METHOD _log : BOOL
  VAR_INPUT
    {attribute 'TcHmiSymbol.Show'}
    name : STRING;  (* Name of this function block instance *)
  END_VAR
  VAR_IN_OUT
    {attribute 'TcHmiSymbol.Show'}
    buffer : LogBuffer;  (* Buffer to write all logging to *)
  END_VAR
  VAR
    {attribute 'TcHmiSymbol.Show'}
    subBuffer : LogBuffer;  (* Temporary buffer to write logging by parts (sub-statemachines) to *)
  END_VAR
                  THIS^.processes.setEnabled._log(
    name := 'processes.setEnabled',
    buffer := subBuffer);
LOGGER(
    name := name,
    actualStatus := THIS^.actualStatus,
    previousStatus := THIS^.previousStatus,
    buffer := buffer,
    subBuffer := subBuffer,
    pBusyStatus := ADR(THIS^.statuses.busyStatus));

                
END_METHOD
END_FUNCTION_BLOCK

FUNCTION_BLOCK SM_ConfigManager
  VAR_INPUT
    {attribute 'TcHmiSymbol.Show'}
    {attribute 'OPC.UA.DA' := '1'}
    {attribute 'OPC.UA.DA.Access' := '1'}
    filePath : STRING;  (* Full path of the config filename *)
    {attribute 'TcHmiSymbol.Show'}
    {attribute 'OPC.UA.DA' := '0'}
    {attribute 'TcHmiSymbol.Hide'}
    isEnabled : BOOL;  (* Is control enabled? *)
  END_VAR
  VAR_OUTPUT
    {attribute 'OPC.UA.DA' := '1'}
    {attribute 'OPC.UA.DA.Access' := '1'}
    {attribute 'TcHmiSymbol.Show'}
    actualStatus : STRING;  (* Current status description *)
    {attribute 'TcHmiSymbol.Show'}
    previousStatus : STRING;  (* Previous status description *)
    {attribute 'TcHmiSymbol.Show'}
    statuses : ConfigManagerStatuses;  (* Statuses of the state machine *)
    {attribute 'TcHmiSymbol.Show'}
    processes : ConfigManagerProcesses;  (* Processes of the state machine *)
  END_VAR

            statuses.busyStatus( isBusy := processes.save.statuses.busyStatus.busy OR (processes.load.statuses.busyStatus.busy OR processes.activate.statuses.busyStatus.busy) );
statuses.healthStatus(
    isGood := processes.save.statuses.healthStatus.isGood AND (processes.load.statuses.healthStatus.isGood AND processes.activate.statuses.healthStatus.isGood),
    hasWarning := processes.save.statuses.healthStatus.hasWarning OR (processes.load.statuses.healthStatus.hasWarning OR processes.activate.statuses.healthStatus.hasWarning));
processes.save( isEnabled := isEnabled AND statuses.busyStatus.idle );
processes.load( isEnabled := isEnabled AND statuses.busyStatus.idle );
processes.activate( isEnabled := isEnabled AND statuses.busyStatus.idle );

          

{attribute 'TcRpcEnable' := '1'}
METHOD save : RequestResults
  VAR_INPUT
    {attribute 'TcHmiSymbol.Show'}
    filePath : STRING;
  END_VAR
                  save := THIS^.processes.save.request( filePath := filePath );

                
END_METHOD

{attribute 'TcRpcEnable' := '1'}
METHOD load : RequestResults
  VAR_INPUT
    {attribute 'TcHmiSymbol.Show'}
    filePath : STRING;
  END_VAR
                  load := THIS^.processes.load.request( filePath := filePath );

                
END_METHOD

{attribute 'TcRpcEnable' := '1'}
METHOD activate : RequestResults
                  activate := THIS^.processes.activate.request();

                
END_METHOD

METHOD _log : BOOL
  VAR_INPUT
    {attribute 'TcHmiSymbol.Show'}
    name : STRING;  (* Name of this function block instance *)
  END_VAR
  VAR_IN_OUT
    {attribute 'TcHmiSymbol.Show'}
    buffer : LogBuffer;  (* Buffer to write all logging to *)
  END_VAR
  VAR
    {attribute 'TcHmiSymbol.Show'}
    subBuffer : LogBuffer;  (* Temporary buffer to write logging by parts (sub-statemachines) to *)
  END_VAR
                  THIS^.processes.save._log(
    name := 'processes.save',
    buffer := subBuffer);
THIS^.processes.load._log(
    name := 'processes.load',
    buffer := subBuffer);
THIS^.processes.activate._log(
    name := 'processes.activate',
    buffer := subBuffer);
LOGGER(
    name := name,
    actualStatus := THIS^.actualStatus,
    previousStatus := THIS^.previousStatus,
    buffer := buffer,
    subBuffer := subBuffer,
    pHealthStatus := ADR(THIS^.statuses.healthStatus),
    pBusyStatus := ADR(THIS^.statuses.busyStatus));

                
END_METHOD
END_FUNCTION_BLOCK

FUNCTION_BLOCK SM_ModbusRTUBus
  VAR_INPUT
    {attribute 'TcHmiSymbol.Show'}
    {attribute 'OPC.UA.DA' := '1'}
    {attribute 'OPC.UA.DA.Access' := '1'}
    retries : INT := 3;  (* Number of retries for a succesfull process *)
    {attribute 'TcHmiSymbol.Show'}
    {attribute 'OPC.UA.DA' := '0'}
    {attribute 'TcHmiSymbol.Hide'}
    isEnabled : BOOL;  (* Is control enabled? *)
  END_VAR
  VAR_OUTPUT
    {attribute 'OPC.UA.DA' := '1'}
    {attribute 'OPC.UA.DA.Access' := '1'}
    {attribute 'TcHmiSymbol.Show'}
    actualStatus : STRING;  (* Current status description *)
    {attribute 'TcHmiSymbol.Show'}
    previousStatus : STRING;  (* Previous status description *)
    {attribute 'TcHmiSymbol.Show'}
    statuses : ModbusRTUBusStatuses;  (* Statuses of the state machine *)
    {attribute 'TcHmiSymbol.Show'}
    processes : ModbusRTUBusProcesses;  (* Processes of the state machine *)
  END_VAR

            statuses.busyStatus( isBusy := processes.readCoil.statuses.busyStatus.busy OR (processes.writeCoil.statuses.busyStatus.busy OR (processes.readRegister.statuses.busyStatus.busy OR (processes.writeRegister.statuses.busyStatus.busy OR processes.diagnostics.statuses.busyStatus.busy))) );
processes.readCoil( isEnabled := isEnabled AND statuses.busyStatus.idle );
processes.writeCoil( isEnabled := isEnabled AND statuses.busyStatus.idle );
processes.readRegister( isEnabled := isEnabled AND statuses.busyStatus.idle );
processes.writeRegister( isEnabled := isEnabled AND statuses.busyStatus.idle );
processes.diagnostics( isEnabled := isEnabled AND statuses.busyStatus.idle );

          

{attribute 'TcRpcEnable' := '1'}
METHOD readCoil : RequestResults
  VAR_INPUT
    {attribute 'TcHmiSymbol.Show'}
    unitID : USINT;
    {attribute 'TcHmiSymbol.Show'}
    address : UINT;
  END_VAR
                  readCoil := THIS^.processes.readCoil.request(
    unitID := unitID,
    address := address);

                
END_METHOD

{attribute 'TcRpcEnable' := '1'}
METHOD writeCoil : RequestResults
  VAR_INPUT
    {attribute 'TcHmiSymbol.Show'}
    unitID : USINT;
    {attribute 'TcHmiSymbol.Show'}
    address : UINT;
    {attribute 'TcHmiSymbol.Show'}
    value : BOOL;
  END_VAR
                  writeCoil := THIS^.processes.writeCoil.request(
    unitID := unitID,
    address := address,
    value := value);

                
END_METHOD

{attribute 'TcRpcEnable' := '1'}
METHOD readRegister : RequestResults
  VAR_INPUT
    {attribute 'TcHmiSymbol.Show'}
    unitID : USINT;
    {attribute 'TcHmiSymbol.Show'}
    address : UINT;
  END_VAR
                  readRegister := THIS^.processes.readRegister.request(
    unitID := unitID,
    address := address);

                
END_METHOD

{attribute 'TcRpcEnable' := '1'}
METHOD writeRegister : RequestResults
  VAR_INPUT
    {attribute 'TcHmiSymbol.Show'}
    unitID : USINT;
    {attribute 'TcHmiSymbol.Show'}
    address : UINT;
    {attribute 'TcHmiSymbol.Show'}
    value : INT;
  END_VAR
                  writeRegister := THIS^.processes.writeRegister.request(
    unitID := unitID,
    address := address,
    value := value);

                
END_METHOD

{attribute 'TcRpcEnable' := '1'}
METHOD diagnostics : RequestResults
  VAR_INPUT
    {attribute 'TcHmiSymbol.Show'}
    unitID : USINT;
    {attribute 'TcHmiSymbol.Show'}
    subFunction : UINT;
    {attribute 'TcHmiSymbol.Show'}
    subData : INT;
  END_VAR
                  diagnostics := THIS^.processes.diagnostics.request(
    unitID := unitID,
    subFunction := subFunction,
    subData := subData);

                
END_METHOD

METHOD _log : BOOL
  VAR_INPUT
    {attribute 'TcHmiSymbol.Show'}
    name : STRING;  (* Name of this function block instance *)
  END_VAR
  VAR_IN_OUT
    {attribute 'TcHmiSymbol.Show'}
    buffer : LogBuffer;  (* Buffer to write all logging to *)
  END_VAR
  VAR
    {attribute 'TcHmiSymbol.Show'}
    subBuffer : LogBuffer;  (* Temporary buffer to write logging by parts (sub-statemachines) to *)
  END_VAR
                  THIS^.processes.readCoil._log(
    name := 'processes.readCoil',
    buffer := subBuffer);
THIS^.processes.writeCoil._log(
    name := 'processes.writeCoil',
    buffer := subBuffer);
THIS^.processes.readRegister._log(
    name := 'processes.readRegister',
    buffer := subBuffer);
THIS^.processes.writeRegister._log(
    name := 'processes.writeRegister',
    buffer := subBuffer);
THIS^.processes.diagnostics._log(
    name := 'processes.diagnostics',
    buffer := subBuffer);
LOGGER(
    name := name,
    actualStatus := THIS^.actualStatus,
    previousStatus := THIS^.previousStatus,
    buffer := buffer,
    subBuffer := subBuffer,
    pBusyStatus := ADR(THIS^.statuses.busyStatus));

                
END_METHOD
END_FUNCTION_BLOCK

FUNCTION_BLOCK Process EXTENDS BaseProcess
  VAR
    {attribute 'OPC.UA.DA' := '0'}
    testVar : BOOL;  (* At least 1 variable needed because subclass members of an empty class are not exposed by OPC UA (TwinCAT bug!) *)
  END_VAR

            IF do_request THEN
    do_request_result := request();
    do_request := FALSE;
END_IF;
SUPER^();

          

{attribute 'TcRpcEnable' := '1'}
METHOD start
                  THIS^.statuses.busyStatus( isBusy := TRUE );
THIS^.statuses.healthStatus( isGood := TRUE );

                
END_METHOD

{attribute 'TcRpcEnable' := '1'}
METHOD request : RequestResults
                  IF THIS^.statuses.enabledStatus.enabled THEN
    request := RequestResults.ACCEPTED;
    THIS^.start();
ELSE
    request := RequestResults.REJECTED;
END_IF;

                
END_METHOD
END_FUNCTION_BLOCK

FUNCTION_BLOCK McProcess EXTENDS BaseMcProcess
  VAR
    {attribute 'OPC.UA.DA' := '0'}
    testVar : BOOL;  (* At least 1 variable needed because subclass members of an empty class are not exposed by OPC UA (TwinCAT bug!) *)
  END_VAR

            IF do_request THEN
    do_request_result := request();
    do_request := FALSE;
END_IF;
SUPER^();

          

{attribute 'TcRpcEnable' := '1'}
METHOD start
                  THIS^.statuses.busyStatus( isBusy := TRUE );
THIS^.statuses.healthStatus( isGood := TRUE );

                
END_METHOD

{attribute 'TcRpcEnable' := '1'}
METHOD request : RequestResults
                  IF THIS^.statuses.enabledStatus.enabled THEN
    request := RequestResults.ACCEPTED;
    THIS^.start();
ELSE
    request := RequestResults.REJECTED;
END_IF;

                
END_METHOD
END_FUNCTION_BLOCK

FUNCTION_BLOCK ChangeSetpointProcess EXTENDS BaseProcess
  VAR_INPUT
    {attribute 'OPC.UA.DA' := '1'}
    {attribute 'TcHmiSymbol.Show'}
    set : ChangeSetpointProcessArgs;  (* Arguments to be set, before writing do_request TRUE *)
  END_VAR
  VAR_OUTPUT
    {attribute 'OPC.UA.DA' := '1'}
    {attribute 'OPC.UA.DA.Access' := '1'}
    {attribute 'TcHmiSymbol.Show'}
    get : ChangeSetpointProcessArgs;  (* Arguments in use by the process, if do_request was accepted *)
  END_VAR

            IF do_request THEN
    do_request_result := request( setpoint := set.setpoint );
    do_request := FALSE;
END_IF;
SUPER^();

          

{attribute 'TcRpcEnable' := '1'}
METHOD start
  VAR_INPUT
    {attribute 'TcHmiSymbol.Show'}
    setpoint : LREAL;  (* New setpoint value *)
  END_VAR
                  THIS^.get.setpoint := setpoint;
THIS^.statuses.busyStatus( isBusy := TRUE );
THIS^.statuses.healthStatus( isGood := TRUE );

                
END_METHOD

{attribute 'TcRpcEnable' := '1'}
METHOD request : RequestResults
  VAR_INPUT
    {attribute 'TcHmiSymbol.Show'}
    setpoint : LREAL;  (* New setpoint value *)
  END_VAR
                  IF THIS^.statuses.enabledStatus.enabled THEN
    request := RequestResults.ACCEPTED;
    THIS^.start( setpoint := setpoint );
ELSE
    request := RequestResults.REJECTED;
END_IF;

                
END_METHOD
END_FUNCTION_BLOCK

FUNCTION_BLOCK ChangeParameterProcess EXTENDS BaseProcess
  VAR_INPUT
    {attribute 'OPC.UA.DA' := '1'}
    {attribute 'TcHmiSymbol.Show'}
    set : ChangeParameterProcessArgs;  (* Arguments to be set, before writing do_request TRUE *)
  END_VAR
  VAR_OUTPUT
    {attribute 'OPC.UA.DA' := '1'}
    {attribute 'OPC.UA.DA.Access' := '1'}
    {attribute 'TcHmiSymbol.Show'}
    get : ChangeParameterProcessArgs;  (* Arguments in use by the process, if do_request was accepted *)
  END_VAR

            IF do_request THEN
    do_request_result := request( parameter := set.parameter );
    do_request := FALSE;
END_IF;
SUPER^();

          

{attribute 'TcRpcEnable' := '1'}
METHOD start
  VAR_INPUT
    {attribute 'TcHmiSymbol.Show'}
    parameter : LREAL;  (* New parameter value *)
  END_VAR
                  THIS^.get.parameter := parameter;
THIS^.statuses.busyStatus( isBusy := TRUE );
THIS^.statuses.healthStatus( isGood := TRUE );

                
END_METHOD

{attribute 'TcRpcEnable' := '1'}
METHOD request : RequestResults
  VAR_INPUT
    {attribute 'TcHmiSymbol.Show'}
    parameter : LREAL;  (* New parameter value *)
  END_VAR
                  IF THIS^.statuses.enabledStatus.enabled THEN
    request := RequestResults.ACCEPTED;
    THIS^.start( parameter := parameter );
ELSE
    request := RequestResults.REJECTED;
END_IF;

                
END_METHOD
END_FUNCTION_BLOCK

FUNCTION_BLOCK McMoveAbsoluteProcess EXTENDS BaseMcProcess
  VAR_INPUT
    {attribute 'OPC.UA.DA' := '1'}
    {attribute 'TcHmiSymbol.Show'}
    set : McMoveAbsoluteProcessArgs;  (* Arguments to be set, before writing do_request TRUE *)
  END_VAR
  VAR_OUTPUT
    {attribute 'OPC.UA.DA' := '1'}
    {attribute 'OPC.UA.DA.Access' := '1'}
    {attribute 'TcHmiSymbol.Show'}
    get : McMoveAbsoluteProcessArgs;  (* Arguments in use by the process, if do_request was accepted *)
  END_VAR

            IF do_request THEN
    do_request_result := request(
    position := set.position,
    maxVelocity := set.maxVelocity);
    do_request := FALSE;
END_IF;
SUPER^();

          

{attribute 'TcRpcEnable' := '1'}
METHOD start
  VAR_INPUT
    {attribute 'TcHmiSymbol.Show'}
    position : LREAL;  (* New position setpoint *)
    {attribute 'TcHmiSymbol.Show'}
    maxVelocity : LREAL;  (* Maximum velocity *)
  END_VAR
                  THIS^.get.position := position;
THIS^.get.maxVelocity := maxVelocity;
THIS^.statuses.busyStatus( isBusy := TRUE );
THIS^.statuses.healthStatus( isGood := TRUE );

                
END_METHOD

{attribute 'TcRpcEnable' := '1'}
METHOD request : RequestResults
  VAR_INPUT
    {attribute 'TcHmiSymbol.Show'}
    position : LREAL;  (* New position setpoint *)
    {attribute 'TcHmiSymbol.Show'}
    maxVelocity : LREAL;  (* Maximum velocity *)
  END_VAR
                  IF THIS^.statuses.enabledStatus.enabled THEN
    request := RequestResults.ACCEPTED;
    THIS^.start(
        position := position,
        maxVelocity := maxVelocity);
ELSE
    request := RequestResults.REJECTED;
END_IF;

                
END_METHOD
END_FUNCTION_BLOCK

FUNCTION_BLOCK McMoveRelativeProcess EXTENDS BaseMcProcess
  VAR_INPUT
    {attribute 'OPC.UA.DA' := '1'}
    {attribute 'TcHmiSymbol.Show'}
    set : McMoveRelativeProcessArgs;  (* Arguments to be set, before writing do_request TRUE *)
  END_VAR
  VAR_OUTPUT
    {attribute 'OPC.UA.DA' := '1'}
    {attribute 'OPC.UA.DA.Access' := '1'}
    {attribute 'TcHmiSymbol.Show'}
    get : McMoveRelativeProcessArgs;  (* Arguments in use by the process, if do_request was accepted *)
  END_VAR

            IF do_request THEN
    do_request_result := request(
    distance := set.distance,
    maxVelocity := set.maxVelocity);
    do_request := FALSE;
END_IF;
SUPER^();

          

{attribute 'TcRpcEnable' := '1'}
METHOD start
  VAR_INPUT
    {attribute 'TcHmiSymbol.Show'}
    distance : LREAL;  (* Distance to move *)
    {attribute 'TcHmiSymbol.Show'}
    maxVelocity : LREAL;  (* Maximum velocity *)
  END_VAR
                  THIS^.get.distance := distance;
THIS^.get.maxVelocity := maxVelocity;
THIS^.statuses.busyStatus( isBusy := TRUE );
THIS^.statuses.healthStatus( isGood := TRUE );

                
END_METHOD

{attribute 'TcRpcEnable' := '1'}
METHOD request : RequestResults
  VAR_INPUT
    {attribute 'TcHmiSymbol.Show'}
    distance : LREAL;  (* Distance to move *)
    {attribute 'TcHmiSymbol.Show'}
    maxVelocity : LREAL;  (* Maximum velocity *)
  END_VAR
                  IF THIS^.statuses.enabledStatus.enabled THEN
    request := RequestResults.ACCEPTED;
    THIS^.start(
        distance := distance,
        maxVelocity := maxVelocity);
ELSE
    request := RequestResults.REJECTED;
END_IF;

                
END_METHOD
END_FUNCTION_BLOCK

FUNCTION_BLOCK McPowerProcess EXTENDS BaseMcProcess
  VAR_INPUT
    {attribute 'OPC.UA.DA' := '1'}
    {attribute 'TcHmiSymbol.Show'}
    set : McPowerProcessArgs;  (* Arguments to be set, before writing do_request TRUE *)
  END_VAR
  VAR_OUTPUT
    {attribute 'OPC.UA.DA' := '1'}
    {attribute 'OPC.UA.DA.Access' := '1'}
    {attribute 'TcHmiSymbol.Show'}
    get : McPowerProcessArgs;  (* Arguments in use by the process, if do_request was accepted *)
  END_VAR

            IF do_request THEN
    do_request_result := request( enable := set.enable );
    do_request := FALSE;
END_IF;
SUPER^();

          

{attribute 'TcRpcEnable' := '1'}
METHOD start
  VAR_INPUT
    {attribute 'TcHmiSymbol.Show'}
    enable : BOOL;  (* Enable the power or not *)
  END_VAR
                  THIS^.get.enable := enable;
THIS^.statuses.busyStatus( isBusy := TRUE );
THIS^.statuses.healthStatus( isGood := TRUE );

                
END_METHOD

{attribute 'TcRpcEnable' := '1'}
METHOD request : RequestResults
  VAR_INPUT
    {attribute 'TcHmiSymbol.Show'}
    enable : BOOL;  (* Enable the power or not *)
  END_VAR
                  IF THIS^.statuses.enabledStatus.enabled THEN
    request := RequestResults.ACCEPTED;
    THIS^.start( enable := enable );
ELSE
    request := RequestResults.REJECTED;
END_IF;

                
END_METHOD
END_FUNCTION_BLOCK

FUNCTION_BLOCK McSetPositionProcess EXTENDS BaseMcProcess
  VAR_INPUT
    {attribute 'OPC.UA.DA' := '1'}
    {attribute 'TcHmiSymbol.Show'}
    set : McSetPositionProcessArgs;  (* Arguments to be set, before writing do_request TRUE *)
  END_VAR
  VAR_OUTPUT
    {attribute 'OPC.UA.DA' := '1'}
    {attribute 'OPC.UA.DA.Access' := '1'}
    {attribute 'TcHmiSymbol.Show'}
    get : McSetPositionProcessArgs;  (* Arguments in use by the process, if do_request was accepted *)
  END_VAR

            IF do_request THEN
    do_request_result := request( value := set.value );
    do_request := FALSE;
END_IF;
SUPER^();

          

{attribute 'TcRpcEnable' := '1'}
METHOD start
  VAR_INPUT
    {attribute 'TcHmiSymbol.Show'}
    value : LREAL;  (* New position to be taken over by the encoder *)
  END_VAR
                  THIS^.get.value := value;
THIS^.statuses.busyStatus( isBusy := TRUE );
THIS^.statuses.healthStatus( isGood := TRUE );

                
END_METHOD

{attribute 'TcRpcEnable' := '1'}
METHOD request : RequestResults
  VAR_INPUT
    {attribute 'TcHmiSymbol.Show'}
    value : LREAL;  (* New position to be taken over by the encoder *)
  END_VAR
                  IF THIS^.statuses.enabledStatus.enabled THEN
    request := RequestResults.ACCEPTED;
    THIS^.start( value := value );
ELSE
    request := RequestResults.REJECTED;
END_IF;

                
END_METHOD
END_FUNCTION_BLOCK

FUNCTION_BLOCK McStopProcess EXTENDS BaseMcProcess
  VAR_INPUT
    {attribute 'OPC.UA.DA' := '1'}
    {attribute 'TcHmiSymbol.Show'}
    set : McStopProcessArgs;  (* Arguments to be set, before writing do_request TRUE *)
  END_VAR
  VAR_OUTPUT
    {attribute 'OPC.UA.DA' := '1'}
    {attribute 'OPC.UA.DA.Access' := '1'}
    {attribute 'TcHmiSymbol.Show'}
    get : McStopProcessArgs;  (* Arguments in use by the process, if do_request was accepted *)
  END_VAR

            IF do_request THEN
    do_request_result := request(
    deceleration := set.deceleration,
    jerk := set.jerk);
    do_request := FALSE;
END_IF;
SUPER^();

          

{attribute 'TcRpcEnable' := '1'}
METHOD start
  VAR_INPUT
    {attribute 'TcHmiSymbol.Show'}
    deceleration : LREAL;  (* Deceleration (use 0 for default). If non zero, then also jerk must be non zero! *)
    {attribute 'TcHmiSymbol.Show'}
    jerk : LREAL;  (* Jerk (use 0 for default). If non zero, then also deceleration must be non zero! *)
  END_VAR
                  THIS^.get.deceleration := deceleration;
THIS^.get.jerk := jerk;
THIS^.statuses.busyStatus( isBusy := TRUE );
THIS^.statuses.healthStatus( isGood := TRUE );

                
END_METHOD

{attribute 'TcRpcEnable' := '1'}
METHOD request : RequestResults
  VAR_INPUT
    {attribute 'TcHmiSymbol.Show'}
    deceleration : LREAL;  (* Deceleration (use 0 for default). If non zero, then also jerk must be non zero! *)
    {attribute 'TcHmiSymbol.Show'}
    jerk : LREAL;  (* Jerk (use 0 for default). If non zero, then also deceleration must be non zero! *)
  END_VAR
                  IF THIS^.statuses.enabledStatus.enabled THEN
    request := RequestResults.ACCEPTED;
    THIS^.start(
        deceleration := deceleration,
        jerk := jerk);
ELSE
    request := RequestResults.REJECTED;
END_IF;

                
END_METHOD
END_FUNCTION_BLOCK

FUNCTION_BLOCK McMoveVelocityProcess EXTENDS BaseMcProcess
  VAR_INPUT
    {attribute 'OPC.UA.DA' := '1'}
    {attribute 'TcHmiSymbol.Show'}
    set : McMoveVelocityProcessArgs;  (* Arguments to be set, before writing do_request TRUE *)
  END_VAR
  VAR_OUTPUT
    {attribute 'OPC.UA.DA' := '1'}
    {attribute 'OPC.UA.DA.Access' := '1'}
    {attribute 'TcHmiSymbol.Show'}
    get : McMoveVelocityProcessArgs;  (* Arguments in use by the process, if do_request was accepted *)
  END_VAR

            IF do_request THEN
    do_request_result := request( value := set.value );
    do_request := FALSE;
END_IF;
SUPER^();

          

{attribute 'TcRpcEnable' := '1'}
METHOD start
  VAR_INPUT
    {attribute 'TcHmiSymbol.Show'}
    value : LREAL;  (* New velocity *)
  END_VAR
                  THIS^.get.value := value;
THIS^.statuses.busyStatus( isBusy := TRUE );
THIS^.statuses.healthStatus( isGood := TRUE );

                
END_METHOD

{attribute 'TcRpcEnable' := '1'}
METHOD request : RequestResults
  VAR_INPUT
    {attribute 'TcHmiSymbol.Show'}
    value : LREAL;  (* New velocity *)
  END_VAR
                  IF THIS^.statuses.enabledStatus.enabled THEN
    request := RequestResults.ACCEPTED;
    THIS^.start( value := value );
ELSE
    request := RequestResults.REJECTED;
END_IF;

                
END_METHOD
END_FUNCTION_BLOCK

FUNCTION_BLOCK SetEnabledProcess EXTENDS BaseProcess
  VAR_INPUT
    {attribute 'OPC.UA.DA' := '1'}
    {attribute 'TcHmiSymbol.Show'}
    set : SetEnabledProcessArgs;  (* Arguments to be set, before writing do_request TRUE *)
  END_VAR
  VAR_OUTPUT
    {attribute 'OPC.UA.DA' := '1'}
    {attribute 'OPC.UA.DA.Access' := '1'}
    {attribute 'TcHmiSymbol.Show'}
    get : SetEnabledProcessArgs;  (* Arguments in use by the process, if do_request was accepted *)
  END_VAR

            IF do_request THEN
    do_request_result := request( enabled := set.enabled );
    do_request := FALSE;
END_IF;
SUPER^();

          

{attribute 'TcRpcEnable' := '1'}
METHOD start
  VAR_INPUT
    {attribute 'TcHmiSymbol.Show'}
    enabled : BOOL;  (* True to enable, false to disable *)
  END_VAR
                  THIS^.get.enabled := enabled;
THIS^.statuses.busyStatus( isBusy := TRUE );
THIS^.statuses.healthStatus( isGood := TRUE );

                
END_METHOD

{attribute 'TcRpcEnable' := '1'}
METHOD request : RequestResults
  VAR_INPUT
    {attribute 'TcHmiSymbol.Show'}
    enabled : BOOL;  (* True to enable, false to disable *)
  END_VAR
                  IF THIS^.statuses.enabledStatus.enabled THEN
    request := RequestResults.ACCEPTED;
    THIS^.start( enabled := enabled );
ELSE
    request := RequestResults.REJECTED;
END_IF;

                
END_METHOD
END_FUNCTION_BLOCK

FUNCTION_BLOCK McWriteParameter EXTENDS BaseMcProcess
  VAR_INPUT
    {attribute 'OPC.UA.DA' := '1'}
    {attribute 'TcHmiSymbol.Show'}
    set : McWriteParameterArgs;  (* Arguments to be set, before writing do_request TRUE *)
  END_VAR
  VAR_OUTPUT
    {attribute 'OPC.UA.DA' := '1'}
    {attribute 'OPC.UA.DA.Access' := '1'}
    {attribute 'TcHmiSymbol.Show'}
    get : McWriteParameterArgs;  (* Arguments in use by the process, if do_request was accepted *)
  END_VAR

            IF do_request THEN
    do_request_result := request(
    parameterNumber := set.parameterNumber,
    value := set.value);
    do_request := FALSE;
END_IF;
SUPER^();

          

{attribute 'TcRpcEnable' := '1'}
METHOD start
  VAR_INPUT
    {attribute 'TcHmiSymbol.Show'}
    parameterNumber : INT;  (* Number of the parameter *)
    {attribute 'TcHmiSymbol.Show'}
    value : LREAL;  (* Value to write *)
  END_VAR
                  THIS^.get.parameterNumber := parameterNumber;
THIS^.get.value := value;
THIS^.statuses.busyStatus( isBusy := TRUE );
THIS^.statuses.healthStatus( isGood := TRUE );

                
END_METHOD

{attribute 'TcRpcEnable' := '1'}
METHOD request : RequestResults
  VAR_INPUT
    {attribute 'TcHmiSymbol.Show'}
    parameterNumber : INT;  (* Number of the parameter *)
    {attribute 'TcHmiSymbol.Show'}
    value : LREAL;  (* Value to write *)
  END_VAR
                  IF THIS^.statuses.enabledStatus.enabled THEN
    request := RequestResults.ACCEPTED;
    THIS^.start(
        parameterNumber := parameterNumber,
        value := value);
ELSE
    request := RequestResults.REJECTED;
END_IF;

                
END_METHOD
END_FUNCTION_BLOCK

FUNCTION_BLOCK McReadParameter EXTENDS BaseMcProcess
  VAR_INPUT
    {attribute 'TcHmiSymbol.Show'}
    value : LREAL;  (* Value that was read *)
    {attribute 'OPC.UA.DA' := '1'}
    {attribute 'TcHmiSymbol.Show'}
    set : McReadParameterArgs;  (* Arguments to be set, before writing do_request TRUE *)
  END_VAR
  VAR_OUTPUT
    {attribute 'OPC.UA.DA' := '1'}
    {attribute 'OPC.UA.DA.Access' := '1'}
    {attribute 'TcHmiSymbol.Show'}
    get : McReadParameterArgs;  (* Arguments in use by the process, if do_request was accepted *)
  END_VAR

            IF do_request THEN
    do_request_result := request( parameterNumber := set.parameterNumber );
    do_request := FALSE;
END_IF;
SUPER^();

          

{attribute 'TcRpcEnable' := '1'}
METHOD start
  VAR_INPUT
    {attribute 'TcHmiSymbol.Show'}
    parameterNumber : INT;  (* Number of the parameter *)
  END_VAR
                  THIS^.get.parameterNumber := parameterNumber;
THIS^.statuses.busyStatus( isBusy := TRUE );
THIS^.statuses.healthStatus( isGood := TRUE );

                
END_METHOD

{attribute 'TcRpcEnable' := '1'}
METHOD request : RequestResults
  VAR_INPUT
    {attribute 'TcHmiSymbol.Show'}
    parameterNumber : INT;  (* Number of the parameter *)
  END_VAR
                  IF THIS^.statuses.enabledStatus.enabled THEN
    request := RequestResults.ACCEPTED;
    THIS^.start( parameterNumber := parameterNumber );
ELSE
    request := RequestResults.REJECTED;
END_IF;

                
END_METHOD
END_FUNCTION_BLOCK

FUNCTION_BLOCK McWriteBoolParameter EXTENDS BaseMcProcess
  VAR_INPUT
    {attribute 'OPC.UA.DA' := '1'}
    {attribute 'TcHmiSymbol.Show'}
    set : McWriteBoolParameterArgs;  (* Arguments to be set, before writing do_request TRUE *)
  END_VAR
  VAR_OUTPUT
    {attribute 'OPC.UA.DA' := '1'}
    {attribute 'OPC.UA.DA.Access' := '1'}
    {attribute 'TcHmiSymbol.Show'}
    get : McWriteBoolParameterArgs;  (* Arguments in use by the process, if do_request was accepted *)
  END_VAR

            IF do_request THEN
    do_request_result := request(
    parameterNumber := set.parameterNumber,
    value := set.value);
    do_request := FALSE;
END_IF;
SUPER^();

          

{attribute 'TcRpcEnable' := '1'}
METHOD start
  VAR_INPUT
    {attribute 'TcHmiSymbol.Show'}
    parameterNumber : INT;  (* Number of the parameter *)
    {attribute 'TcHmiSymbol.Show'}
    value : BOOL;  (* Value to write *)
  END_VAR
                  THIS^.get.parameterNumber := parameterNumber;
THIS^.get.value := value;
THIS^.statuses.busyStatus( isBusy := TRUE );
THIS^.statuses.healthStatus( isGood := TRUE );

                
END_METHOD

{attribute 'TcRpcEnable' := '1'}
METHOD request : RequestResults
  VAR_INPUT
    {attribute 'TcHmiSymbol.Show'}
    parameterNumber : INT;  (* Number of the parameter *)
    {attribute 'TcHmiSymbol.Show'}
    value : BOOL;  (* Value to write *)
  END_VAR
                  IF THIS^.statuses.enabledStatus.enabled THEN
    request := RequestResults.ACCEPTED;
    THIS^.start(
        parameterNumber := parameterNumber,
        value := value);
ELSE
    request := RequestResults.REJECTED;
END_IF;

                
END_METHOD
END_FUNCTION_BLOCK

FUNCTION_BLOCK McReadBoolParameter EXTENDS BaseMcProcess
  VAR_INPUT
    {attribute 'TcHmiSymbol.Show'}
    value : BOOL;  (* Value that was read *)
    {attribute 'OPC.UA.DA' := '1'}
    {attribute 'TcHmiSymbol.Show'}
    set : McReadBoolParameterArgs;  (* Arguments to be set, before writing do_request TRUE *)
  END_VAR
  VAR_OUTPUT
    {attribute 'OPC.UA.DA' := '1'}
    {attribute 'OPC.UA.DA.Access' := '1'}
    {attribute 'TcHmiSymbol.Show'}
    get : McReadBoolParameterArgs;  (* Arguments in use by the process, if do_request was accepted *)
  END_VAR

            IF do_request THEN
    do_request_result := request( parameterNumber := set.parameterNumber );
    do_request := FALSE;
END_IF;
SUPER^();

          

{attribute 'TcRpcEnable' := '1'}
METHOD start
  VAR_INPUT
    {attribute 'TcHmiSymbol.Show'}
    parameterNumber : INT;  (* Number of the parameter *)
  END_VAR
                  THIS^.get.parameterNumber := parameterNumber;
THIS^.statuses.busyStatus( isBusy := TRUE );
THIS^.statuses.healthStatus( isGood := TRUE );

                
END_METHOD

{attribute 'TcRpcEnable' := '1'}
METHOD request : RequestResults
  VAR_INPUT
    {attribute 'TcHmiSymbol.Show'}
    parameterNumber : INT;  (* Number of the parameter *)
  END_VAR
                  IF THIS^.statuses.enabledStatus.enabled THEN
    request := RequestResults.ACCEPTED;
    THIS^.start( parameterNumber := parameterNumber );
ELSE
    request := RequestResults.REJECTED;
END_IF;

                
END_METHOD
END_FUNCTION_BLOCK

FUNCTION_BLOCK McProbe EXTENDS BaseMcProcess
  VAR_INPUT
    {attribute 'TcHmiSymbol.Show'}
    recordedPosition : LREAL;  (* Value that was probed *)
    {attribute 'OPC.UA.DA' := '1'}
    {attribute 'TcHmiSymbol.Show'}
    set : McProbeArgs;  (* Arguments to be set, before writing do_request TRUE *)
  END_VAR
  VAR_OUTPUT
    {attribute 'OPC.UA.DA' := '1'}
    {attribute 'OPC.UA.DA.Access' := '1'}
    {attribute 'TcHmiSymbol.Show'}
    get : McProbeArgs;  (* Arguments in use by the process, if do_request was accepted *)
  END_VAR

            IF do_request THEN
    do_request_result := request(
    risingEdge := set.risingEdge,
    timeout := set.timeout);
    do_request := FALSE;
END_IF;
SUPER^();

          

{attribute 'TcRpcEnable' := '1'}
METHOD start
  VAR_INPUT
    {attribute 'TcHmiSymbol.Show'}
    risingEdge : BOOL;  (* True to probe the rising edge, false to probe the falling edge *)
    {attribute 'TcHmiSymbol.Show'}
    timeout : LREAL;  (* Timeout, in seconds. After this timeout, probing is aborted. timeout <= 0 means endless probing. *)
  END_VAR
                  THIS^.get.risingEdge := risingEdge;
THIS^.get.timeout := timeout;
THIS^.statuses.busyStatus( isBusy := TRUE );
THIS^.statuses.healthStatus( isGood := TRUE );

                
END_METHOD

{attribute 'TcRpcEnable' := '1'}
METHOD request : RequestResults
  VAR_INPUT
    {attribute 'TcHmiSymbol.Show'}
    risingEdge : BOOL;  (* True to probe the rising edge, false to probe the falling edge *)
    {attribute 'TcHmiSymbol.Show'}
    timeout : LREAL;  (* Timeout, in seconds. After this timeout, probing is aborted. timeout <= 0 means endless probing. *)
  END_VAR
                  IF THIS^.statuses.enabledStatus.enabled THEN
    request := RequestResults.ACCEPTED;
    THIS^.start(
        risingEdge := risingEdge,
        timeout := timeout);
ELSE
    request := RequestResults.REJECTED;
END_IF;

                
END_METHOD
END_FUNCTION_BLOCK

FUNCTION_BLOCK SDOReadProcess EXTENDS BaseProcess
  VAR_INPUT
    {attribute 'TcHmiSymbol.Show'}
    value1Byte : USINT;  (* Value that has been read, if noOfBytes is 1 *)
    {attribute 'TcHmiSymbol.Show'}
    value2Bytes : UINT;  (* Value that has been read, if noOfBytes is 2 *)
    {attribute 'TcHmiSymbol.Show'}
    value4Bytes : UDINT;  (* Value that has been read, if noOfBytes is 4 *)
    {attribute 'TcHmiSymbol.Show'}
    errorId : UDINT;  (* Error ID according to Beckhoff *)
    {attribute 'OPC.UA.DA' := '1'}
    {attribute 'TcHmiSymbol.Show'}
    set : SDOReadProcessArgs;  (* Arguments to be set, before writing do_request TRUE *)
  END_VAR
  VAR_OUTPUT
    {attribute 'OPC.UA.DA' := '1'}
    {attribute 'OPC.UA.DA.Access' := '1'}
    {attribute 'TcHmiSymbol.Show'}
    get : SDOReadProcessArgs;  (* Arguments in use by the process, if do_request was accepted *)
  END_VAR

            IF do_request THEN
    do_request_result := request(
    index := set.index,
    subindex := set.subindex,
    noOfBytes := set.noOfBytes);
    do_request := FALSE;
END_IF;
SUPER^();

          

{attribute 'TcRpcEnable' := '1'}
METHOD start
  VAR_INPUT
    {attribute 'TcHmiSymbol.Show'}
    index : UINT;  (* SDO Index *)
    {attribute 'TcHmiSymbol.Show'}
    subindex : USINT;  (* SDO SubIndex *)
    {attribute 'TcHmiSymbol.Show'}
    noOfBytes : UDINT;  (* Number of bytes to be read *)
  END_VAR
                  THIS^.get.index := index;
THIS^.get.subindex := subindex;
THIS^.get.noOfBytes := noOfBytes;
THIS^.statuses.busyStatus( isBusy := TRUE );
THIS^.statuses.healthStatus( isGood := TRUE );

                
END_METHOD

{attribute 'TcRpcEnable' := '1'}
METHOD request : RequestResults
  VAR_INPUT
    {attribute 'TcHmiSymbol.Show'}
    index : UINT;  (* SDO Index *)
    {attribute 'TcHmiSymbol.Show'}
    subindex : USINT;  (* SDO SubIndex *)
    {attribute 'TcHmiSymbol.Show'}
    noOfBytes : UDINT;  (* Number of bytes to be read *)
  END_VAR
                  IF THIS^.statuses.enabledStatus.enabled THEN
    request := RequestResults.ACCEPTED;
    THIS^.start(
        index := index,
        subindex := subindex,
        noOfBytes := noOfBytes);
ELSE
    request := RequestResults.REJECTED;
END_IF;

                
END_METHOD
END_FUNCTION_BLOCK

FUNCTION_BLOCK SDOWriteProcess EXTENDS BaseProcess
  VAR_INPUT
    {attribute 'TcHmiSymbol.Show'}
    errorId : UDINT;  (* Error ID according to Beckhoff *)
    {attribute 'OPC.UA.DA' := '1'}
    {attribute 'TcHmiSymbol.Show'}
    set : SDOWriteProcessArgs;  (* Arguments to be set, before writing do_request TRUE *)
  END_VAR
  VAR_OUTPUT
    {attribute 'OPC.UA.DA' := '1'}
    {attribute 'OPC.UA.DA.Access' := '1'}
    {attribute 'TcHmiSymbol.Show'}
    get : SDOWriteProcessArgs;  (* Arguments in use by the process, if do_request was accepted *)
  END_VAR

            IF do_request THEN
    do_request_result := request(
    index := set.index,
    subindex := set.subindex,
    noOfBytes := set.noOfBytes,
    value1Byte := set.value1Byte,
    value2Bytes := set.value2Bytes,
    value4Bytes := set.value4Bytes);
    do_request := FALSE;
END_IF;
SUPER^();

          

{attribute 'TcRpcEnable' := '1'}
METHOD start
  VAR_INPUT
    {attribute 'TcHmiSymbol.Show'}
    index : UINT;  (* SDO Index *)
    {attribute 'TcHmiSymbol.Show'}
    subindex : USINT;  (* SDO SubIndex *)
    {attribute 'TcHmiSymbol.Show'}
    noOfBytes : UDINT;  (* Number of bytes to be written *)
    {attribute 'TcHmiSymbol.Show'}
    value1Byte : USINT;  (* Value to be written if noOfBytes is 1 *)
    {attribute 'TcHmiSymbol.Show'}
    value2Bytes : UINT;  (* Value to be written if noOfBytes is 2 *)
    {attribute 'TcHmiSymbol.Show'}
    value4Bytes : UDINT;  (* Value to be written if noOfBytes is 4 *)
  END_VAR
                  THIS^.get.index := index;
THIS^.get.subindex := subindex;
THIS^.get.noOfBytes := noOfBytes;
THIS^.get.value1Byte := value1Byte;
THIS^.get.value2Bytes := value2Bytes;
THIS^.get.value4Bytes := value4Bytes;
THIS^.statuses.busyStatus( isBusy := TRUE );
THIS^.statuses.healthStatus( isGood := TRUE );

                
END_METHOD

{attribute 'TcRpcEnable' := '1'}
METHOD request : RequestResults
  VAR_INPUT
    {attribute 'TcHmiSymbol.Show'}
    index : UINT;  (* SDO Index *)
    {attribute 'TcHmiSymbol.Show'}
    subindex : USINT;  (* SDO SubIndex *)
    {attribute 'TcHmiSymbol.Show'}
    noOfBytes : UDINT;  (* Number of bytes to be written *)
    {attribute 'TcHmiSymbol.Show'}
    value1Byte : USINT;  (* Value to be written if noOfBytes is 1 *)
    {attribute 'TcHmiSymbol.Show'}
    value2Bytes : UINT;  (* Value to be written if noOfBytes is 2 *)
    {attribute 'TcHmiSymbol.Show'}
    value4Bytes : UDINT;  (* Value to be written if noOfBytes is 4 *)
  END_VAR
                  IF THIS^.statuses.enabledStatus.enabled THEN
    request := RequestResults.ACCEPTED;
    THIS^.start(
        index := index,
        subindex := subindex,
        noOfBytes := noOfBytes,
        value1Byte := value1Byte,
        value2Bytes := value2Bytes,
        value4Bytes := value4Bytes);
ELSE
    request := RequestResults.REJECTED;
END_IF;

                
END_METHOD
END_FUNCTION_BLOCK

FUNCTION_BLOCK SoEReadProcess EXTENDS BaseProcess
  VAR_INPUT
    {attribute 'TcHmiSymbol.Show'}
    value1Byte : USINT;  (* Value that has been read, if noOfBytes is 1 *)
    {attribute 'TcHmiSymbol.Show'}
    value2Bytes : UINT;  (* Value that has been read, if noOfBytes is 2 *)
    {attribute 'TcHmiSymbol.Show'}
    value4Bytes : UDINT;  (* Value that has been read, if noOfBytes is 4 *)
    {attribute 'TcHmiSymbol.Show'}
    adsErrorId : UINT;  (* ADS error ID *)
    {attribute 'TcHmiSymbol.Show'}
    sercosErrorId : UINT;  (* Sercos error ID *)
    {attribute 'OPC.UA.DA' := '1'}
    {attribute 'TcHmiSymbol.Show'}
    set : SoEReadProcessArgs;  (* Arguments to be set, before writing do_request TRUE *)
  END_VAR
  VAR_OUTPUT
    {attribute 'OPC.UA.DA' := '1'}
    {attribute 'OPC.UA.DA.Access' := '1'}
    {attribute 'TcHmiSymbol.Show'}
    get : SoEReadProcessArgs;  (* Arguments in use by the process, if do_request was accepted *)
  END_VAR

            IF do_request THEN
    do_request_result := request(
    index := set.index,
    noOfBytes := set.noOfBytes);
    do_request := FALSE;
END_IF;
SUPER^();

          

{attribute 'TcRpcEnable' := '1'}
METHOD start
  VAR_INPUT
    {attribute 'TcHmiSymbol.Show'}
    index : UINT;  (* SDO Index *)
    {attribute 'TcHmiSymbol.Show'}
    noOfBytes : UDINT;  (* Number of bytes to be read *)
  END_VAR
                  THIS^.get.index := index;
THIS^.get.noOfBytes := noOfBytes;
THIS^.statuses.busyStatus( isBusy := TRUE );
THIS^.statuses.healthStatus( isGood := TRUE );

                
END_METHOD

{attribute 'TcRpcEnable' := '1'}
METHOD request : RequestResults
  VAR_INPUT
    {attribute 'TcHmiSymbol.Show'}
    index : UINT;  (* SDO Index *)
    {attribute 'TcHmiSymbol.Show'}
    noOfBytes : UDINT;  (* Number of bytes to be read *)
  END_VAR
                  IF THIS^.statuses.enabledStatus.enabled THEN
    request := RequestResults.ACCEPTED;
    THIS^.start(
        index := index,
        noOfBytes := noOfBytes);
ELSE
    request := RequestResults.REJECTED;
END_IF;

                
END_METHOD
END_FUNCTION_BLOCK

FUNCTION_BLOCK SoEWriteProcess EXTENDS BaseProcess
  VAR_INPUT
    {attribute 'TcHmiSymbol.Show'}
    adsErrorId : UINT;  (* ADS error ID *)
    {attribute 'TcHmiSymbol.Show'}
    sercosErrorId : UINT;  (* Sercos error ID *)
    {attribute 'OPC.UA.DA' := '1'}
    {attribute 'TcHmiSymbol.Show'}
    set : SoEWriteProcessArgs;  (* Arguments to be set, before writing do_request TRUE *)
  END_VAR
  VAR_OUTPUT
    {attribute 'OPC.UA.DA' := '1'}
    {attribute 'OPC.UA.DA.Access' := '1'}
    {attribute 'TcHmiSymbol.Show'}
    get : SoEWriteProcessArgs;  (* Arguments in use by the process, if do_request was accepted *)
  END_VAR

            IF do_request THEN
    do_request_result := request(
    index := set.index,
    noOfBytes := set.noOfBytes,
    value1Byte := set.value1Byte,
    value2Bytes := set.value2Bytes,
    value4Bytes := set.value4Bytes);
    do_request := FALSE;
END_IF;
SUPER^();

          

{attribute 'TcRpcEnable' := '1'}
METHOD start
  VAR_INPUT
    {attribute 'TcHmiSymbol.Show'}
    index : UINT;  (* SDO Index *)
    {attribute 'TcHmiSymbol.Show'}
    noOfBytes : UDINT;  (* Number of bytes to be written *)
    {attribute 'TcHmiSymbol.Show'}
    value1Byte : USINT;  (* Value to be written if noOfBytes is 1 *)
    {attribute 'TcHmiSymbol.Show'}
    value2Bytes : UINT;  (* Value to be written if noOfBytes is 2 *)
    {attribute 'TcHmiSymbol.Show'}
    value4Bytes : UDINT;  (* Value to be written if noOfBytes is 4 *)
  END_VAR
                  THIS^.get.index := index;
THIS^.get.noOfBytes := noOfBytes;
THIS^.get.value1Byte := value1Byte;
THIS^.get.value2Bytes := value2Bytes;
THIS^.get.value4Bytes := value4Bytes;
THIS^.statuses.busyStatus( isBusy := TRUE );
THIS^.statuses.healthStatus( isGood := TRUE );

                
END_METHOD

{attribute 'TcRpcEnable' := '1'}
METHOD request : RequestResults
  VAR_INPUT
    {attribute 'TcHmiSymbol.Show'}
    index : UINT;  (* SDO Index *)
    {attribute 'TcHmiSymbol.Show'}
    noOfBytes : UDINT;  (* Number of bytes to be written *)
    {attribute 'TcHmiSymbol.Show'}
    value1Byte : USINT;  (* Value to be written if noOfBytes is 1 *)
    {attribute 'TcHmiSymbol.Show'}
    value2Bytes : UINT;  (* Value to be written if noOfBytes is 2 *)
    {attribute 'TcHmiSymbol.Show'}
    value4Bytes : UDINT;  (* Value to be written if noOfBytes is 4 *)
  END_VAR
                  IF THIS^.statuses.enabledStatus.enabled THEN
    request := RequestResults.ACCEPTED;
    THIS^.start(
        index := index,
        noOfBytes := noOfBytes,
        value1Byte := value1Byte,
        value2Bytes := value2Bytes,
        value4Bytes := value4Bytes);
ELSE
    request := RequestResults.REJECTED;
END_IF;

                
END_METHOD
END_FUNCTION_BLOCK

FUNCTION_BLOCK SoEResetProcess EXTENDS BaseProcess
  VAR_INPUT
    {attribute 'TcHmiSymbol.Show'}
    adsErrorId : UINT;  (* ADS error ID *)
    {attribute 'TcHmiSymbol.Show'}
    sercosErrorId : UINT;  (* Sercos error ID *)
  END_VAR

            IF do_request THEN
    do_request_result := request();
    do_request := FALSE;
END_IF;
SUPER^();

          

{attribute 'TcRpcEnable' := '1'}
METHOD start
                  THIS^.statuses.busyStatus( isBusy := TRUE );
THIS^.statuses.healthStatus( isGood := TRUE );

                
END_METHOD

{attribute 'TcRpcEnable' := '1'}
METHOD request : RequestResults
                  IF THIS^.statuses.enabledStatus.enabled THEN
    request := RequestResults.ACCEPTED;
    THIS^.start();
ELSE
    request := RequestResults.REJECTED;
END_IF;

                
END_METHOD
END_FUNCTION_BLOCK

FUNCTION_BLOCK SetBrakeProcess EXTENDS BaseProcess
  VAR_INPUT
    {attribute 'OPC.UA.DA' := '1'}
    {attribute 'TcHmiSymbol.Show'}
    set : SetBrakeProcessArgs;  (* Arguments to be set, before writing do_request TRUE *)
  END_VAR
  VAR_OUTPUT
    {attribute 'OPC.UA.DA' := '1'}
    {attribute 'OPC.UA.DA.Access' := '1'}
    {attribute 'TcHmiSymbol.Show'}
    get : SetBrakeProcessArgs;  (* Arguments in use by the process, if do_request was accepted *)
  END_VAR

            IF do_request THEN
    do_request_result := request( newState := set.newState );
    do_request := FALSE;
END_IF;
SUPER^();

          

{attribute 'TcRpcEnable' := '1'}
METHOD start
  VAR_INPUT
    {attribute 'TcHmiSymbol.Show'}
    newState : DriveBrakeStates;  (* Requested brake state *)
  END_VAR
                  THIS^.get.newState := newState;
THIS^.statuses.busyStatus( isBusy := TRUE );
THIS^.statuses.healthStatus( isGood := TRUE );

                
END_METHOD

{attribute 'TcRpcEnable' := '1'}
METHOD request : RequestResults
  VAR_INPUT
    {attribute 'TcHmiSymbol.Show'}
    newState : DriveBrakeStates;  (* Requested brake state *)
  END_VAR
                  IF THIS^.statuses.enabledStatus.enabled THEN
    request := RequestResults.ACCEPTED;
    THIS^.start( newState := newState );
ELSE
    request := RequestResults.REJECTED;
END_IF;

                
END_METHOD
END_FUNCTION_BLOCK

FUNCTION_BLOCK ChangeOperatingStateProcess EXTENDS BaseProcess
  VAR_INPUT
    {attribute 'OPC.UA.DA' := '1'}
    {attribute 'TcHmiSymbol.Show'}
    set : ChangeOperatingStateProcessArgs;  (* Arguments to be set, before writing do_request TRUE *)
  END_VAR
  VAR_OUTPUT
    {attribute 'OPC.UA.DA' := '1'}
    {attribute 'OPC.UA.DA.Access' := '1'}
    {attribute 'TcHmiSymbol.Show'}
    get : ChangeOperatingStateProcessArgs;  (* Arguments in use by the process, if do_request was accepted *)
  END_VAR

            IF do_request THEN
    do_request_result := request( state := set.state );
    do_request := FALSE;
END_IF;
SUPER^();

          

{attribute 'TcRpcEnable' := '1'}
METHOD start
  VAR_INPUT
    {attribute 'TcHmiSymbol.Show'}
    state : OperatingStates;  (* New operating state (e.g. AUTO, MANUAL) *)
  END_VAR
                  THIS^.get.state := state;
THIS^.statuses.busyStatus( isBusy := TRUE );
THIS^.statuses.healthStatus( isGood := TRUE );

                
END_METHOD

{attribute 'TcRpcEnable' := '1'}
METHOD request : RequestResults
  VAR_INPUT
    {attribute 'TcHmiSymbol.Show'}
    state : OperatingStates;  (* New operating state (e.g. AUTO, MANUAL) *)
  END_VAR
                  IF THIS^.statuses.enabledStatus.enabled THEN
    request := RequestResults.ACCEPTED;
    THIS^.start( state := state );
ELSE
    request := RequestResults.REJECTED;
END_IF;

                
END_METHOD
END_FUNCTION_BLOCK

FUNCTION_BLOCK ChangeOperatorStateProcess EXTENDS BaseProcess
  VAR_INPUT
    {attribute 'OPC.UA.DA' := '1'}
    {attribute 'TcHmiSymbol.Show'}
    set : ChangeOperatorStateProcessArgs;  (* Arguments to be set, before writing do_request TRUE *)
  END_VAR
  VAR_OUTPUT
    {attribute 'OPC.UA.DA' := '1'}
    {attribute 'OPC.UA.DA.Access' := '1'}
    {attribute 'TcHmiSymbol.Show'}
    get : ChangeOperatorStateProcessArgs;  (* Arguments in use by the process, if do_request was accepted *)
  END_VAR

            IF do_request THEN
    do_request_result := request(
    state := set.state,
    password := set.password);
    do_request := FALSE;
END_IF;
SUPER^();

          

{attribute 'TcRpcEnable' := '1'}
METHOD start
  VAR_INPUT
    {attribute 'TcHmiSymbol.Show'}
    state : OperatorStates;  (* New operator state (e.g. OBSERVER, TECH, ...) *)
    {attribute 'TcHmiSymbol.Show'}
    password : STRING;  (* Password (only sometimes required, e.g. to go from OBSERVER to TECH) *)
  END_VAR
                  THIS^.get.state := state;
THIS^.get.password := password;
THIS^.statuses.busyStatus( isBusy := TRUE );
THIS^.statuses.healthStatus( isGood := TRUE );

                
END_METHOD

{attribute 'TcRpcEnable' := '1'}
METHOD request : RequestResults
  VAR_INPUT
    {attribute 'TcHmiSymbol.Show'}
    state : OperatorStates;  (* New operator state (e.g. OBSERVER, TECH, ...) *)
    {attribute 'TcHmiSymbol.Show'}
    password : STRING;  (* Password (only sometimes required, e.g. to go from OBSERVER to TECH) *)
  END_VAR
                  IF THIS^.statuses.enabledStatus.enabled THEN
    request := RequestResults.ACCEPTED;
    THIS^.start(
        state := state,
        password := password);
ELSE
    request := RequestResults.REJECTED;
END_IF;

                
END_METHOD
END_FUNCTION_BLOCK

FUNCTION_BLOCK ChangeOperatingModeStateProcess EXTENDS BaseProcess
  VAR_INPUT
    {attribute 'OPC.UA.DA' := '1'}
    {attribute 'TcHmiSymbol.Show'}
    set : ChangeOperatingModeStateProcessArgs;  (* Arguments to be set, before writing do_request TRUE *)
  END_VAR
  VAR_OUTPUT
    {attribute 'OPC.UA.DA' := '1'}
    {attribute 'OPC.UA.DA.Access' := '1'}
    {attribute 'TcHmiSymbol.Show'}
    get : ChangeOperatingModeStateProcessArgs;  (* Arguments in use by the process, if do_request was accepted *)
  END_VAR

            IF do_request THEN
    do_request_result := request( state := set.state );
    do_request := FALSE;
END_IF;
SUPER^();

          

{attribute 'TcRpcEnable' := '1'}
METHOD start
  VAR_INPUT
    {attribute 'TcHmiSymbol.Show'}
    state : OperatingModeStates;  (* New operating state (e.g. LOCAL, REMOTE) *)
  END_VAR
                  THIS^.get.state := state;
THIS^.statuses.busyStatus( isBusy := TRUE );
THIS^.statuses.healthStatus( isGood := TRUE );

                
END_METHOD

{attribute 'TcRpcEnable' := '1'}
METHOD request : RequestResults
  VAR_INPUT
    {attribute 'TcHmiSymbol.Show'}
    state : OperatingModeStates;  (* New operating state (e.g. LOCAL, REMOTE) *)
  END_VAR
                  IF THIS^.statuses.enabledStatus.enabled THEN
    request := RequestResults.ACCEPTED;
    THIS^.start( state := state );
ELSE
    request := RequestResults.REJECTED;
END_IF;

                
END_METHOD
END_FUNCTION_BLOCK

FUNCTION_BLOCK ReadXmlProcess EXTENDS BaseXmlDataSrvProcess
  VAR_INPUT
    {attribute 'OPC.UA.DA' := '1'}
    {attribute 'TcHmiSymbol.Show'}
    set : ReadXmlProcessArgs;  (* Arguments to be set, before writing do_request TRUE *)
  END_VAR
  VAR_OUTPUT
    {attribute 'OPC.UA.DA' := '1'}
    {attribute 'OPC.UA.DA.Access' := '1'}
    {attribute 'TcHmiSymbol.Show'}
    get : ReadXmlProcessArgs;  (* Arguments in use by the process, if do_request was accepted *)
  END_VAR

            IF do_request THEN
    do_request_result := request( filePath := set.filePath );
    do_request := FALSE;
END_IF;
SUPER^();

          

{attribute 'TcRpcEnable' := '1'}
METHOD start
  VAR_INPUT
    {attribute 'TcHmiSymbol.Show'}
    filePath : STRING;  (* Full path of the filename to read *)
  END_VAR
                  THIS^.get.filePath := filePath;
THIS^.statuses.busyStatus( isBusy := TRUE );
THIS^.statuses.healthStatus( isGood := TRUE );

                
END_METHOD

{attribute 'TcRpcEnable' := '1'}
METHOD request : RequestResults
  VAR_INPUT
    {attribute 'TcHmiSymbol.Show'}
    filePath : STRING;  (* Full path of the filename to read *)
  END_VAR
                  IF THIS^.statuses.enabledStatus.enabled THEN
    request := RequestResults.ACCEPTED;
    THIS^.start( filePath := filePath );
ELSE
    request := RequestResults.REJECTED;
END_IF;

                
END_METHOD
END_FUNCTION_BLOCK

FUNCTION_BLOCK WriteXmlProcess EXTENDS BaseXmlDataSrvProcess
  VAR_INPUT
    {attribute 'OPC.UA.DA' := '1'}
    {attribute 'TcHmiSymbol.Show'}
    set : WriteXmlProcessArgs;  (* Arguments to be set, before writing do_request TRUE *)
  END_VAR
  VAR_OUTPUT
    {attribute 'OPC.UA.DA' := '1'}
    {attribute 'OPC.UA.DA.Access' := '1'}
    {attribute 'TcHmiSymbol.Show'}
    get : WriteXmlProcessArgs;  (* Arguments in use by the process, if do_request was accepted *)
  END_VAR

            IF do_request THEN
    do_request_result := request( filePath := set.filePath );
    do_request := FALSE;
END_IF;
SUPER^();

          

{attribute 'TcRpcEnable' := '1'}
METHOD start
  VAR_INPUT
    {attribute 'TcHmiSymbol.Show'}
    filePath : STRING;  (* Full path of the filename to write *)
  END_VAR
                  THIS^.get.filePath := filePath;
THIS^.statuses.busyStatus( isBusy := TRUE );
THIS^.statuses.healthStatus( isGood := TRUE );

                
END_METHOD

{attribute 'TcRpcEnable' := '1'}
METHOD request : RequestResults
  VAR_INPUT
    {attribute 'TcHmiSymbol.Show'}
    filePath : STRING;  (* Full path of the filename to write *)
  END_VAR
                  IF THIS^.statuses.enabledStatus.enabled THEN
    request := RequestResults.ACCEPTED;
    THIS^.start( filePath := filePath );
ELSE
    request := RequestResults.REJECTED;
END_IF;

                
END_METHOD
END_FUNCTION_BLOCK

FUNCTION_BLOCK ActivateProcess EXTENDS BaseProcess
  VAR
    {attribute 'OPC.UA.DA' := '0'}
    testVar : BOOL;  (* At least 1 variable needed because subclass members of an empty class are not exposed by OPC UA (TwinCAT bug!) *)
  END_VAR

            IF do_request THEN
    do_request_result := request();
    do_request := FALSE;
END_IF;
SUPER^();

          

{attribute 'TcRpcEnable' := '1'}
METHOD start
                  THIS^.statuses.busyStatus( isBusy := TRUE );
THIS^.statuses.healthStatus( isGood := TRUE );

                
END_METHOD

{attribute 'TcRpcEnable' := '1'}
METHOD request : RequestResults
                  IF THIS^.statuses.enabledStatus.enabled THEN
    request := RequestResults.ACCEPTED;
    THIS^.start();
ELSE
    request := RequestResults.REJECTED;
END_IF;

                
END_METHOD
END_FUNCTION_BLOCK

FUNCTION_BLOCK ModbusRTUBusReadCoilProcess EXTENDS BaseProcess
  VAR_INPUT
    {attribute 'TcHmiSymbol.Show'}
    value : BOOL;  (* Value of the coil *)
    {attribute 'TcHmiSymbol.Show'}
    errorId : INT;  (* Error Id. Modbus error code *)
    {attribute 'OPC.UA.DA' := '1'}
    {attribute 'TcHmiSymbol.Show'}
    set : ModbusRTUBusReadCoilProcessArgs;  (* Arguments to be set, before writing do_request TRUE *)
  END_VAR
  VAR_OUTPUT
    {attribute 'OPC.UA.DA' := '1'}
    {attribute 'OPC.UA.DA.Access' := '1'}
    {attribute 'TcHmiSymbol.Show'}
    get : ModbusRTUBusReadCoilProcessArgs;  (* Arguments in use by the process, if do_request was accepted *)
  END_VAR

            IF do_request THEN
    do_request_result := request(
    unitID := set.unitID,
    address := set.address);
    do_request := FALSE;
END_IF;
SUPER^();

          

{attribute 'TcRpcEnable' := '1'}
METHOD start
  VAR_INPUT
    {attribute 'TcHmiSymbol.Show'}
    unitID : USINT;  (* Modbus station address (1..247) *)
    {attribute 'TcHmiSymbol.Show'}
    address : UINT;  (* Modbus data address *)
  END_VAR
                  THIS^.get.unitID := unitID;
THIS^.get.address := address;
THIS^.statuses.busyStatus( isBusy := TRUE );
THIS^.statuses.healthStatus( isGood := TRUE );

                
END_METHOD

{attribute 'TcRpcEnable' := '1'}
METHOD request : RequestResults
  VAR_INPUT
    {attribute 'TcHmiSymbol.Show'}
    unitID : USINT;  (* Modbus station address (1..247) *)
    {attribute 'TcHmiSymbol.Show'}
    address : UINT;  (* Modbus data address *)
  END_VAR
                  IF THIS^.statuses.enabledStatus.enabled THEN
    request := RequestResults.ACCEPTED;
    THIS^.start(
        unitID := unitID,
        address := address);
ELSE
    request := RequestResults.REJECTED;
END_IF;

                
END_METHOD
END_FUNCTION_BLOCK

FUNCTION_BLOCK ModbusRTUBusWriteCoilProcess EXTENDS BaseProcess
  VAR_INPUT
    {attribute 'TcHmiSymbol.Show'}
    errorId : INT;  (* Error Id. Modbus error code *)
    {attribute 'OPC.UA.DA' := '1'}
    {attribute 'TcHmiSymbol.Show'}
    set : ModbusRTUBusWriteCoilProcessArgs;  (* Arguments to be set, before writing do_request TRUE *)
  END_VAR
  VAR_OUTPUT
    {attribute 'OPC.UA.DA' := '1'}
    {attribute 'OPC.UA.DA.Access' := '1'}
    {attribute 'TcHmiSymbol.Show'}
    get : ModbusRTUBusWriteCoilProcessArgs;  (* Arguments in use by the process, if do_request was accepted *)
  END_VAR

            IF do_request THEN
    do_request_result := request(
    unitID := set.unitID,
    address := set.address,
    value := set.value);
    do_request := FALSE;
END_IF;
SUPER^();

          

{attribute 'TcRpcEnable' := '1'}
METHOD start
  VAR_INPUT
    {attribute 'TcHmiSymbol.Show'}
    unitID : USINT;  (* Modbus station address (1..247) *)
    {attribute 'TcHmiSymbol.Show'}
    address : UINT;  (* Modbus data address *)
    {attribute 'TcHmiSymbol.Show'}
    value : BOOL;  (* Value to write on the coil *)
  END_VAR
                  THIS^.get.unitID := unitID;
THIS^.get.address := address;
THIS^.get.value := value;
THIS^.statuses.busyStatus( isBusy := TRUE );
THIS^.statuses.healthStatus( isGood := TRUE );

                
END_METHOD

{attribute 'TcRpcEnable' := '1'}
METHOD request : RequestResults
  VAR_INPUT
    {attribute 'TcHmiSymbol.Show'}
    unitID : USINT;  (* Modbus station address (1..247) *)
    {attribute 'TcHmiSymbol.Show'}
    address : UINT;  (* Modbus data address *)
    {attribute 'TcHmiSymbol.Show'}
    value : BOOL;  (* Value to write on the coil *)
  END_VAR
                  IF THIS^.statuses.enabledStatus.enabled THEN
    request := RequestResults.ACCEPTED;
    THIS^.start(
        unitID := unitID,
        address := address,
        value := value);
ELSE
    request := RequestResults.REJECTED;
END_IF;

                
END_METHOD
END_FUNCTION_BLOCK

FUNCTION_BLOCK ModbusRTUBusReadRegisterProcess EXTENDS BaseProcess
  VAR_INPUT
    {attribute 'TcHmiSymbol.Show'}
    value : INT;  (* Value of the register *)
    {attribute 'TcHmiSymbol.Show'}
    errorId : INT;  (* Error Id. Modbus error code *)
    {attribute 'OPC.UA.DA' := '1'}
    {attribute 'TcHmiSymbol.Show'}
    set : ModbusRTUBusReadRegisterProcessArgs;  (* Arguments to be set, before writing do_request TRUE *)
  END_VAR
  VAR_OUTPUT
    {attribute 'OPC.UA.DA' := '1'}
    {attribute 'OPC.UA.DA.Access' := '1'}
    {attribute 'TcHmiSymbol.Show'}
    get : ModbusRTUBusReadRegisterProcessArgs;  (* Arguments in use by the process, if do_request was accepted *)
  END_VAR

            IF do_request THEN
    do_request_result := request(
    unitID := set.unitID,
    address := set.address);
    do_request := FALSE;
END_IF;
SUPER^();

          

{attribute 'TcRpcEnable' := '1'}
METHOD start
  VAR_INPUT
    {attribute 'TcHmiSymbol.Show'}
    unitID : USINT;  (* Modbus station address (1..247) *)
    {attribute 'TcHmiSymbol.Show'}
    address : UINT;  (* Modbus data address *)
  END_VAR
                  THIS^.get.unitID := unitID;
THIS^.get.address := address;
THIS^.statuses.busyStatus( isBusy := TRUE );
THIS^.statuses.healthStatus( isGood := TRUE );

                
END_METHOD

{attribute 'TcRpcEnable' := '1'}
METHOD request : RequestResults
  VAR_INPUT
    {attribute 'TcHmiSymbol.Show'}
    unitID : USINT;  (* Modbus station address (1..247) *)
    {attribute 'TcHmiSymbol.Show'}
    address : UINT;  (* Modbus data address *)
  END_VAR
                  IF THIS^.statuses.enabledStatus.enabled THEN
    request := RequestResults.ACCEPTED;
    THIS^.start(
        unitID := unitID,
        address := address);
ELSE
    request := RequestResults.REJECTED;
END_IF;

                
END_METHOD
END_FUNCTION_BLOCK

FUNCTION_BLOCK ModbusRTUBusWriteRegisterProcess EXTENDS BaseProcess
  VAR_INPUT
    {attribute 'TcHmiSymbol.Show'}
    errorId : INT;  (* Error Id. Modbus error code *)
    {attribute 'OPC.UA.DA' := '1'}
    {attribute 'TcHmiSymbol.Show'}
    set : ModbusRTUBusWriteRegisterProcessArgs;  (* Arguments to be set, before writing do_request TRUE *)
  END_VAR
  VAR_OUTPUT
    {attribute 'OPC.UA.DA' := '1'}
    {attribute 'OPC.UA.DA.Access' := '1'}
    {attribute 'TcHmiSymbol.Show'}
    get : ModbusRTUBusWriteRegisterProcessArgs;  (* Arguments in use by the process, if do_request was accepted *)
  END_VAR

            IF do_request THEN
    do_request_result := request(
    unitID := set.unitID,
    address := set.address,
    value := set.value);
    do_request := FALSE;
END_IF;
SUPER^();

          

{attribute 'TcRpcEnable' := '1'}
METHOD start
  VAR_INPUT
    {attribute 'TcHmiSymbol.Show'}
    unitID : USINT;  (* Modbus station address (1..247) *)
    {attribute 'TcHmiSymbol.Show'}
    address : UINT;  (* Modbus data address *)
    {attribute 'TcHmiSymbol.Show'}
    value : INT;  (* Value to write on the register *)
  END_VAR
                  THIS^.get.unitID := unitID;
THIS^.get.address := address;
THIS^.get.value := value;
THIS^.statuses.busyStatus( isBusy := TRUE );
THIS^.statuses.healthStatus( isGood := TRUE );

                
END_METHOD

{attribute 'TcRpcEnable' := '1'}
METHOD request : RequestResults
  VAR_INPUT
    {attribute 'TcHmiSymbol.Show'}
    unitID : USINT;  (* Modbus station address (1..247) *)
    {attribute 'TcHmiSymbol.Show'}
    address : UINT;  (* Modbus data address *)
    {attribute 'TcHmiSymbol.Show'}
    value : INT;  (* Value to write on the register *)
  END_VAR
                  IF THIS^.statuses.enabledStatus.enabled THEN
    request := RequestResults.ACCEPTED;
    THIS^.start(
        unitID := unitID,
        address := address,
        value := value);
ELSE
    request := RequestResults.REJECTED;
END_IF;

                
END_METHOD
END_FUNCTION_BLOCK

FUNCTION_BLOCK ModbusRTUBusDiagnosticsProcess EXTENDS BaseProcess
  VAR_INPUT
    {attribute 'TcHmiSymbol.Show'}
    value : INT;  (* Value of the register *)
    {attribute 'TcHmiSymbol.Show'}
    errorId : INT;  (* Error Id. Modbus error code *)
    {attribute 'OPC.UA.DA' := '1'}
    {attribute 'TcHmiSymbol.Show'}
    set : ModbusRTUBusDiagnosticsProcessArgs;  (* Arguments to be set, before writing do_request TRUE *)
  END_VAR
  VAR_OUTPUT
    {attribute 'OPC.UA.DA' := '1'}
    {attribute 'OPC.UA.DA.Access' := '1'}
    {attribute 'TcHmiSymbol.Show'}
    get : ModbusRTUBusDiagnosticsProcessArgs;  (* Arguments in use by the process, if do_request was accepted *)
  END_VAR

            IF do_request THEN
    do_request_result := request(
    unitID := set.unitID,
    subFunction := set.subFunction,
    subData := set.subData);
    do_request := FALSE;
END_IF;
SUPER^();

          

{attribute 'TcRpcEnable' := '1'}
METHOD start
  VAR_INPUT
    {attribute 'TcHmiSymbol.Show'}
    unitID : USINT;  (* Modbus station address (1..247) *)
    {attribute 'TcHmiSymbol.Show'}
    subFunction : UINT;  (* Modbus subFunction code *)
    {attribute 'TcHmiSymbol.Show'}
    subData : INT;  (* Modbus data for subFunction *)
  END_VAR
                  THIS^.get.unitID := unitID;
THIS^.get.subFunction := subFunction;
THIS^.get.subData := subData;
THIS^.statuses.busyStatus( isBusy := TRUE );
THIS^.statuses.healthStatus( isGood := TRUE );

                
END_METHOD

{attribute 'TcRpcEnable' := '1'}
METHOD request : RequestResults
  VAR_INPUT
    {attribute 'TcHmiSymbol.Show'}
    unitID : USINT;  (* Modbus station address (1..247) *)
    {attribute 'TcHmiSymbol.Show'}
    subFunction : UINT;  (* Modbus subFunction code *)
    {attribute 'TcHmiSymbol.Show'}
    subData : INT;  (* Modbus data for subFunction *)
  END_VAR
                  IF THIS^.statuses.enabledStatus.enabled THEN
    request := RequestResults.ACCEPTED;
    THIS^.start(
        unitID := unitID,
        subFunction := subFunction,
        subData := subData);
ELSE
    request := RequestResults.REJECTED;
END_IF;

                
END_METHOD
END_FUNCTION_BLOCK
